FUNCTION_BLOCK CalamityValveBasic (* Basic Function Block Type *)
  (* Standard: 61499-2 *)
  (* Version 0.0, 6/26/2026, Schneider Electric, Template *)
  PACKAGE SE.Nereda;
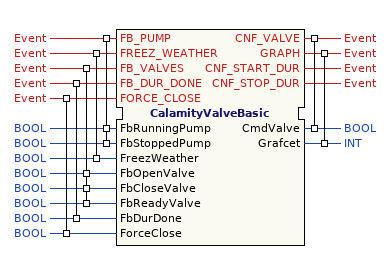
  EVENT_INPUT
    FB_PUMP WITH FbRunningPump, FbStoppedPump; (* Normal Execution Request *)
    FREEZ_WEATHER WITH FreezWeather;
    FB_VALVES WITH FbOpenValve, FbCloseValve, FbReadyValve;
    FB_DUR_DONE WITH FbDurDone;
    FORCE_CLOSE WITH ForceClose;
  END_EVENT
  EVENT_OUTPUT
    CNF_VALVE WITH CmdValve; (* Execution Confirmation *)
    GRAPH WITH Grafcet;
    CNF_START_DUR;
    CNF_STOP_DUR;
  END_EVENT
  VAR_INPUT
    FbRunningPump : BOOL;
    FbStoppedPump : BOOL;
    FreezWeather : BOOL;
    FbOpenValve : BOOL;
    FbCloseValve : BOOL;
    FbReadyValve : BOOL;
    FbDurDone : BOOL;
    ForceClose : BOOL;
  END_VAR
  VAR_OUTPUT
    CmdValve : BOOL;
    Grafcet : INT;
  END_VAR
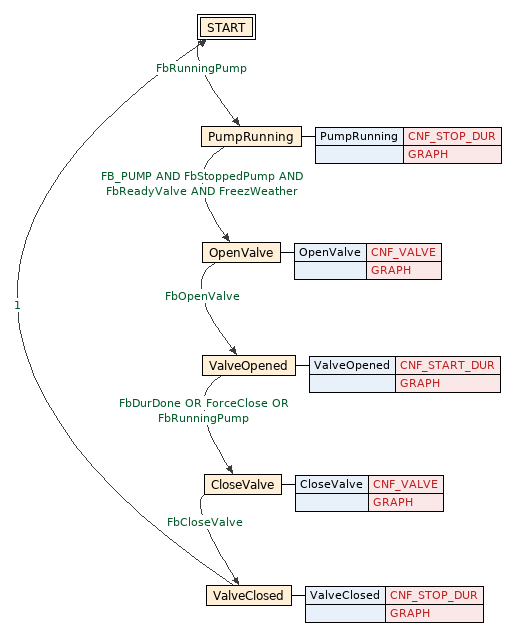
  EC_STATES
    START; (* Initial State *)
    PumpRunning : PumpRunning -> CNF_STOP_DUR, -> GRAPH;
    OpenValve : OpenValve -> CNF_VALVE, -> GRAPH;
    ValveOpened : ValveOpened -> CNF_START_DUR, -> GRAPH;
    CloseValve : CloseValve -> CNF_VALVE, -> GRAPH;
    ValveClosed : ValveClosed -> CNF_STOP_DUR, -> GRAPH;
  END_STATES
  EC_TRANSITIONS
    START TO PumpRunning := FbRunningPump;
    PumpRunning TO OpenValve := FB_PUMP AND FbStoppedPump AND FbReadyValve AND FreezWeather;
    OpenValve TO ValveOpened := FbOpenValve;
    ValveOpened TO CloseValve := FbDurDone OR ForceClose OR FbRunningPump;
    ValveClosed TO START := 1;
    CloseValve TO ValveClosed := FbCloseValve;
  END_TRANSITIONS
  ALGORITHM INIT IN ST: (* Initialization algorithm *)
;
  END_ALGORITHM
  ALGORITHM REQ IN ST: (* Normally executed algorithm *)
;
  END_ALGORITHM
  ALGORITHM OpenValve IN ST:
;
CmdValve := TRUE;
Grafcet := 2;
  END_ALGORITHM
  ALGORITHM CloseValve IN ST:
;
CmdValve := FALSE;
Grafcet := 4;
  END_ALGORITHM
  ALGORITHM ValveOpened IN ST:
;
Grafcet := 3;
  END_ALGORITHM
  ALGORITHM PumpRunning IN ST:
;
Grafcet := 1;
  END_ALGORITHM
  ALGORITHM ValveClosed IN ST:
;
Grafcet := 5;
  END_ALGORITHM
END_FUNCTION_BLOCK
